PROGRAM Main
VAR		
    M1: DUT_MotionStage:=(nCommand:=3); // Yup
	M2: DUT_MotionStage:=(nCommand:=3); // Ydwn
	M3: DUT_MotionStage:=(nCommand:=3); // Xup
	M4: DUT_MotionStage:=(nCommand:=3); // Xdwn
	M5: DUT_MotionStage:=(nCommand:=3); // PitchCoarse
	M6: DUT_MotionStage:=(nCommand:=3); // Bender

	M1_Extras : DUT_MotionStage_Extras;
	M2_Extras : DUT_MotionStage_Extras;
	M3_Extras : DUT_MotionStage_Extras;
	M4_Extras : DUT_MotionStage_Extras;
	M5_Extras : DUT_MotionStage_Extras;
	M6_Extras : DUT_MotionStage_Extras;

	fbMotionStage_x_up, fbMotionStage_x_dwn, fbMotionStage_y_up, fbMotionStage_y_dwn, fbMotionStage_pitch, fbMotionStage_bender : FB_MotionStage;

	bSTOEnable1 AT %I* : BOOL;
	bSTOEnable2 AT %I* : BOOL;
	x_up_enc  AT %I*: ST_RenishawAbsEnc;
	x_dwn_enc  AT %I*: ST_RenishawAbsEnc;
	y_up_enc  AT %I*: ST_RenishawAbsEnc;
	y_dwn_enc  AT %I*: ST_RenishawAbsEnc;

	// Auto coupling function block
	fbAutoCoupleX : FB_GantryAutoCoupling;
	fbAutoCoupleY : FB_GantryAutoCoupling;
	bExecuteCoupleX : BOOL;
	bExecuteCoupleY : BOOL;
	bExecuteDecoupleX : BOOL;
	bExecuteDecoupleY : BOOL;
	bGantryAlreadyCoupledX : BOOL;
	bGantryAlreadyCoupledY : BOOL;
	
	// Gantry variables
	nCurrGantryX : LINT;
	nCurrGantryY : LINT;
	nGantryTolX : LINT := 50000;
	nGantryTolY : LINT := 50000;
END_VAR

// M2L0
// Buttons to enable motors: write 0 to enable, 2 to disable
M1.nEnableMode; // Yup
M2.nEnableMode; // Ydwn
M3.nEnableMode; // Xup
M4.nEnableMode; // Xdwn
M5.nEnableMode; // PitchCoarse

// Encoder Reference Values: Taken from HOMS_FEE project
// Y Gantry really large, not sure if correct. Using initial motor positions for now:
(*
y_up_enc.Ref := 14897597;
y_dwn_enc.Ref := 14551600;
*)
y_up_enc.Ref := 12959000;
y_dwn_enc.Ref := 15964000;
x_up_enc.Ref := 23972500;
x_dwn_enc.Ref := 24766500;

// Gantry Differences to monitor
nCurrGantryY := ((ULINT_TO_LINT(y_up_enc.Count) - ULINT_TO_LINT(y_up_enc.Ref)) - (ULINT_TO_LINT(y_dwn_enc.Count) - ULINT_TO_LINT(y_dwn_enc.Ref)));
nCurrGantryX := ((ULINT_TO_LINT(x_up_enc.Count) - ULINT_TO_LINT(x_up_enc.Ref)) - (ULINT_TO_LINT(x_dwn_enc.Count) - ULINT_TO_LINT(x_dwn_enc.Ref)));

// E-stop
M1.bHardwareEnable := bSTOEnable1 AND bSTOEnable2;
M2.bHardwareEnable := bSTOEnable1 AND bSTOEnable2;
M3.bHardwareEnable := bSTOEnable1 AND bSTOEnable2;
M4.bHardwareEnable := bSTOEnable1 AND bSTOEnable2;
M5.bHardwareEnable := bSTOEnable1 AND bSTOEnable2;
M6.bHardwareEnable := bSTOEnable1 AND bSTOEnable2;

// Start Autocoupling
fbAutoCoupleX(nGantryTol:=nGantryTolX, Master:=M3, MasterEnc:=x_up_enc, Slave:=M4,
	          SlaveEnc:=x_dwn_enc, bExecuteCouple:=bExecuteCoupleX,
              bExecuteDecouple:=bExecuteDecoupleX,
              bGantryAlreadyCoupled=>bGantryAlreadyCoupledX);

fbAutoCoupleY(nGantryTol:=nGantryTolY, Master:=M1, MasterEnc:=y_up_enc, Slave:=M2,
	          SlaveEnc:=y_dwn_enc, bExecuteCouple:=bExecuteCoupleY,
              bExecuteDecouple:=bExecuteDecoupleY,
			  bGantryAlreadyCoupled=>bGantryAlreadyCoupledY);

fbMotionStage_y_up  (stMotionStage:=M1);
fbMotionStage_y_dwn (stMotionStage:=M2);
fbMotionStage_x_up  (stMotionStage:=M3);
fbMotionStage_x_dwn (stMotionStage:=M4);
fbMotionStage_pitch (stMotionStage:=M5);
fbMotionStage_bender (stMotionStage:=M6);

END_PROGRAM

(* stored: Version 1.1.0.1, ProductVersion 3.1.4022.18
   POU MAIN: Id {d73f6033-1c1a-47a8-be0f-3a700ab10cd1}, SpecialFunc None *)
